// TIA Portal V16 export
// export: Created 2020-03-06T18:52:04.6869857Z, ExportSetting WithDefaults, DisplayName Totally Integrated Automation Portal, DisplayVersion V16, DisplayName TIA Portal Version Control Interface, DisplayVersion V16, DisplayName TIA Portal Openness, DisplayVersion V16, DisplayName TIA Portal Teamcenter Gateway, DisplayVersion V16, DisplayName SINAMICS Startdrive Advanced, DisplayVersion V16 Update 1, DisplayName SINAMICS Startdrive G130, G150, S120, S150, SINAMICS MV, S210, DisplayVersion V16 Update 1, DisplayName SINAMICS Startdrive G110M, G120, G120C, G120D, G120P, DisplayVersion V16 Update 1, DisplayName STEP 7 Professional, DisplayVersion V16, DisplayName STEP 7 Safety, DisplayVersion V16, DisplayName WinCC Professional, DisplayVersion V16
FUNCTION_BLOCK "Median 3RR"   // FB871, LAD
{ S7_Optimized_Access := 'TRUE' }
VERSION : 0.3
// stored: AutoNumber false, IsIECCheckEnabled false, IsRetainMemResEnabled false, MemoryReserve 100, SetENOAutomatically false, UDAEnableTagReadback false
   VAR_INPUT
      V1 { ExternalAccessible := 'False'; ExternalVisible := 'False'; ExternalWritable := 'False'} : Real;   // Value 1 REAL
      V2 { ExternalAccessible := 'False'; ExternalVisible := 'False'; ExternalWritable := 'False'} : Real;   // Value 2 REAL
      V3 { ExternalAccessible := 'False'; ExternalVisible := 'False'; ExternalWritable := 'False'} : Real;   // Value 3 REAL
   END_VAR
   VAR_OUTPUT
      MV { ExternalAccessible := 'False'; ExternalVisible := 'False'; ExternalWritable := 'False'} : Real;   // Middle Value
      DGA { ExternalAccessible := 'False'; ExternalVisible := 'False'; ExternalWritable := 'False'} : Bool;   // Deviation General Alarm
      LGA { ExternalAccessible := 'False'; ExternalVisible := 'False'; ExternalWritable := 'False'} : Bool;   // Limit General Alarm
      Spare { ExternalAccessible := 'False'; ExternalVisible := 'False'; ExternalWritable := 'False'} : Bool;   // Spare
   END_VAR
   VAR
      Config : Struct
         DL : Real;   // Deviation Limit
         GL : Real;   // Global Limit
         GH : Real := 1.0;   // Global Hysteresis
         Limits : Struct
            HH : Real;   // High High
            H : Real;   // High
            L : Real;   // Low
            LL : Real;   // Low Low
         END_STRUCT;
         Hysteresis : Struct
            HH : Real;   // High High
            H : Real;   // High
            L : Real;   // Low
            LL : Real;   // Low Low
         END_STRUCT;
      END_STRUCT;
      Status : Struct
         MV : Real;   // Median Value
         HV : Real;   // Highest Value
         LV : Real;   // Lowest Value
         AV : Real;   // Average Value
         V1D : Real;   // Value 1 Deviation
         V2D : Real;   // Value 2 Deviation
         V3D : Real;   // Value 3 Deviation
         V1MV : Bool;   // Value 1 is the Middle Value
         V2MV : Bool;   // Value 2 is the Middle Value
         V3MV : Bool;   // Value 3 is the Middle Value
      END_STRUCT;
      Alarms : Struct
         VHH : Bool;   // Value High High Alarm
         VH : Bool;   // Value High Alarm
         VL : Bool;   // Value Low Alarm
         VLL : Bool;   // Value Low Low Alarm
         V1OD : Bool;   // Value 1 Over Deviation
         V2OD : Bool;   // Value 2 Over Deviation
         V3OD : Bool;   // Value 3 Over Deviation
      END_STRUCT;
      HHA { ExternalAccessible := 'False'; ExternalVisible := 'False'; ExternalWritable := 'False'} : "HLR";   // High High Alarm
      HA { ExternalAccessible := 'False'; ExternalVisible := 'False'; ExternalWritable := 'False'} : "HLR";   // High Alarm
      LA { ExternalAccessible := 'False'; ExternalVisible := 'False'; ExternalWritable := 'False'} : "LLR";   // Low Alarm
      LLA { ExternalAccessible := 'False'; ExternalVisible := 'False'; ExternalWritable := 'False'} : "LLR";   // Low Low Alarm
      V1DL { ExternalAccessible := 'False'; ExternalVisible := 'False'; ExternalWritable := 'False'} : "HLR";   // Value 1 Deviation Limit
      V2DL { ExternalAccessible := 'False'; ExternalVisible := 'False'; ExternalWritable := 'False'} : "HLR";   // Value 2 Deviation Limit
      V3DL { ExternalAccessible := 'False'; ExternalVisible := 'False'; ExternalWritable := 'False'} : "HLR";   // Value 3 Deviation Limit
   END_VAR
   VAR_TEMP
      ME1 : Real;   // Math Equation 1
      ME2 : Real;   // Math Equation 2
      LDV : Real;   // Lowest Deviation Value
      V1DNA : Real;   // Value 1 Deviation Not Absolute
      V2DNA : Real;   // Value 2 Deviation Not Absolute
      V3DNA : Real;   // Value 3 Deviation Not Absolute
      V1DA : Real;   // Value 1 Deviation Absolute
      V2DA : Real;   // Value 2 Deviation Absolute
      V3DA : Real;   // Value 3 Deviation Absolute
      V1MDA : Real;   // Value 1 Median Deviation Absolute
      V2MDA : Real;   // Value 2 Median Deviation Absolute
      V3MDA : Real;   // Value 3 Median Deviation Absolute
   END_VAR
   VAR_TEMP   // added for the SCL form of the ladder/FBD networks
      _w1 : Bool;
   END_VAR
BEGIN

REGION Network 1: Highest Value
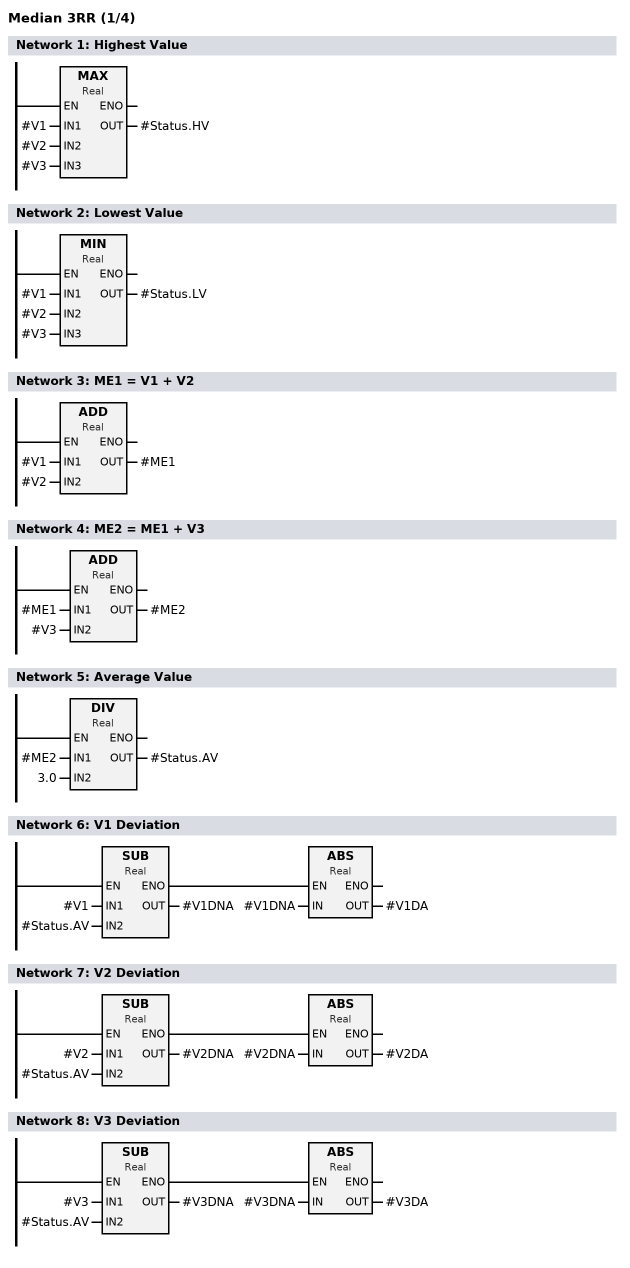
   RUNG wire#powerrail
      { S7_Templates := "[card := 3, value_type := Real]" } MAX(in1 := #V1, in2 := #V2, in3 := #V3, out => #Status.HV)
   END_RUNG
   // the same network as SCL:
   #Status.HV := MAX(IN1 := #V1, IN2 := #V2, IN3 := #V3);
END_REGION

REGION Network 2: Lowest Value
   RUNG wire#powerrail
      { S7_Templates := "[card := 3, value_type := Real]" } MIN(in1 := #V1, in2 := #V2, in3 := #V3, out => #Status.LV)
   END_RUNG
   // the same network as SCL:
   #Status.LV := MIN(IN1 := #V1, IN2 := #V2, IN3 := #V3);
END_REGION

REGION Network 3: ME1 = V1 + V2
   RUNG wire#powerrail
      { S7_Templates := "SrcType := Real"; S7_GenerateENO := "TRUE" } Add(in1 := #V1, in2 := #V2, out => #ME1)
   END_RUNG
   // the same network as SCL:
   #ME1 := #V1 + #V2;
END_REGION

REGION Network 4: ME2 = ME1 + V3
   RUNG wire#powerrail
      { S7_Templates := "SrcType := Real"; S7_GenerateENO := "TRUE" } Add(in1 := #ME1, in2 := #V3, out => #ME2)
   END_RUNG
   // the same network as SCL:
   #ME2 := #ME1 + #V3;
END_REGION

REGION Network 5: Average Value
   RUNG wire#powerrail
      { S7_Templates := "SrcType := Real"; S7_GenerateENO := "TRUE" } Div(in1 := #ME2, in2 := 3.0, out => #Status.AV)
   END_RUNG
   // the same network as SCL:
   #Status.AV := #ME2 / 3.0;
END_REGION

REGION Network 6: V1 Deviation
   RUNG wire#powerrail
      { S7_Templates := "SrcType := Real"; S7_GenerateENO := "TRUE" } Sub(in1 := #V1, in2 := #Status.AV, out => #V1DNA)
      { S7_Templates := "SrcType := Real"; S7_GenerateENO := "TRUE" } Abs(in := #V1DNA, out => #V1DA)
   END_RUNG
   // the same network as SCL:
   // ENO of a box is taken as its EN; it also drops when the box reports an error
   #V1DNA := #V1 - #Status.AV;
   #V1DA := ABS(#V1DNA);
END_REGION

REGION Network 7: V2 Deviation
   RUNG wire#powerrail
      { S7_Templates := "SrcType := Real"; S7_GenerateENO := "TRUE" } Sub(in1 := #V2, in2 := #Status.AV, out => #V2DNA)
      { S7_Templates := "SrcType := Real"; S7_GenerateENO := "TRUE" } Abs(in := #V2DNA, out => #V2DA)
   END_RUNG
   // the same network as SCL:
   // ENO of a box is taken as its EN; it also drops when the box reports an error
   #V2DNA := #V2 - #Status.AV;
   #V2DA := ABS(#V2DNA);
END_REGION

REGION Network 8: V3 Deviation
   RUNG wire#powerrail
      { S7_Templates := "SrcType := Real"; S7_GenerateENO := "TRUE" } Sub(in1 := #V3, in2 := #Status.AV, out => #V3DNA)
      { S7_Templates := "SrcType := Real"; S7_GenerateENO := "TRUE" } Abs(in := #V3DNA, out => #V3DA)
   END_RUNG
   // the same network as SCL:
   // ENO of a box is taken as its EN; it also drops when the box reports an error
   #V3DNA := #V3 - #Status.AV;
   #V3DA := ABS(#V3DNA);
END_REGION

REGION Network 9
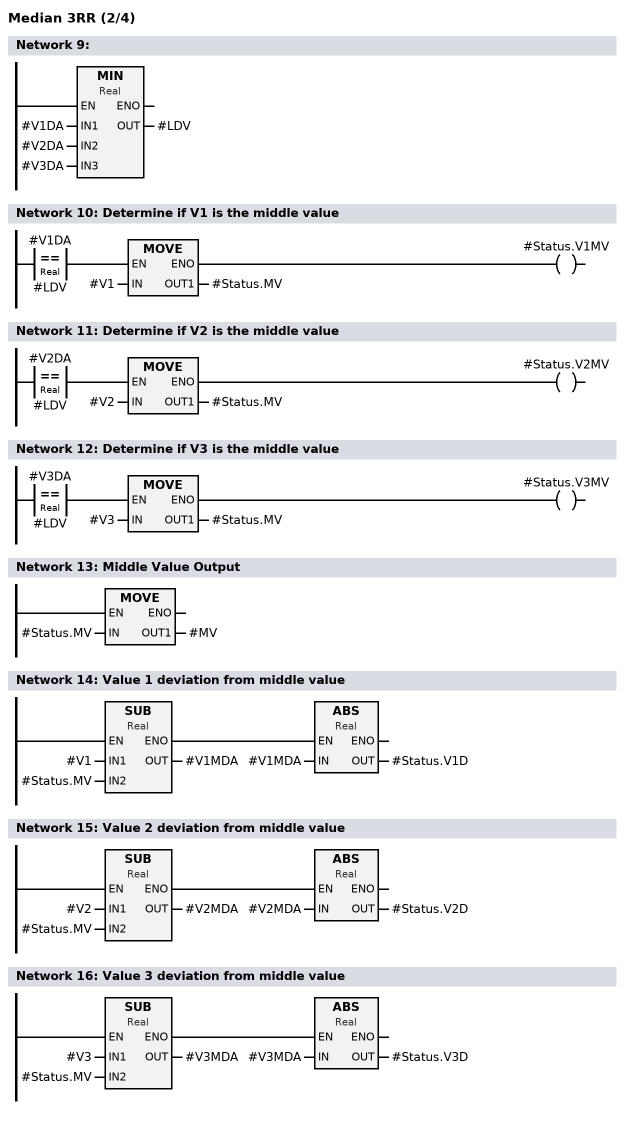
   RUNG wire#powerrail
      { S7_Templates := "[card := 3, value_type := Real]" } MIN(in1 := #V1DA, in2 := #V2DA, in3 := #V3DA, out => #LDV)
   END_RUNG
   // the same network as SCL:
   #LDV := MIN(IN1 := #V1DA, IN2 := #V2DA, IN3 := #V3DA);
END_REGION

REGION Network 10: Determine if V1 is the middle value
   RUNG wire#powerrail
      { S7_Templates := "SrcType := Real" } EQ_Contact(in1 := #V1DA, in2 := #LDV)
      { S7_GenerateENO := "TRUE" } Move(in := #V1, out1 => #Status.MV)
      Coil( #Status.V1MV )
   END_RUNG
   // the same network as SCL:
   // ENO of a box is taken as its EN; it also drops when the box reports an error
   #_w1 := #V1DA = #LDV;
   IF #_w1 THEN #Status.MV := #V1; END_IF;
   #Status.V1MV := #_w1;
END_REGION

REGION Network 11: Determine if V2 is the middle value
   RUNG wire#powerrail
      { S7_Templates := "SrcType := Real" } EQ_Contact(in1 := #V2DA, in2 := #LDV)
      { S7_GenerateENO := "TRUE" } Move(in := #V2, out1 => #Status.MV)
      Coil( #Status.V2MV )
   END_RUNG
   // the same network as SCL:
   // ENO of a box is taken as its EN; it also drops when the box reports an error
   #_w1 := #V2DA = #LDV;
   IF #_w1 THEN #Status.MV := #V2; END_IF;
   #Status.V2MV := #_w1;
END_REGION

REGION Network 12: Determine if V3 is the middle value
   RUNG wire#powerrail
      { S7_Templates := "SrcType := Real" } EQ_Contact(in1 := #V3DA, in2 := #LDV)
      { S7_GenerateENO := "TRUE" } Move(in := #V3, out1 => #Status.MV)
      Coil( #Status.V3MV )
   END_RUNG
   // the same network as SCL:
   // ENO of a box is taken as its EN; it also drops when the box reports an error
   #_w1 := #V3DA = #LDV;
   IF #_w1 THEN #Status.MV := #V3; END_IF;
   #Status.V3MV := #_w1;
END_REGION

REGION Network 13: Middle Value Output
   RUNG wire#powerrail
      { S7_GenerateENO := "TRUE" } Move(in := #Status.MV, out1 => #MV)
   END_RUNG
   // the same network as SCL:
   #MV := #Status.MV;
END_REGION

REGION Network 14: Value 1 deviation from middle value
   RUNG wire#powerrail
      { S7_Templates := "SrcType := Real"; S7_GenerateENO := "TRUE" } Sub(in1 := #V1, in2 := #Status.MV, out => #V1MDA)
      { S7_Templates := "SrcType := Real"; S7_GenerateENO := "TRUE" } Abs(in := #V1MDA, out => #Status.V1D)
   END_RUNG
   // the same network as SCL:
   // ENO of a box is taken as its EN; it also drops when the box reports an error
   #V1MDA := #V1 - #Status.MV;
   #Status.V1D := ABS(#V1MDA);
END_REGION

REGION Network 15: Value 2 deviation from middle value
   RUNG wire#powerrail
      { S7_Templates := "SrcType := Real"; S7_GenerateENO := "TRUE" } Sub(in1 := #V2, in2 := #Status.MV, out => #V2MDA)
      { S7_Templates := "SrcType := Real"; S7_GenerateENO := "TRUE" } Abs(in := #V2MDA, out => #Status.V2D)
   END_RUNG
   // the same network as SCL:
   // ENO of a box is taken as its EN; it also drops when the box reports an error
   #V2MDA := #V2 - #Status.MV;
   #Status.V2D := ABS(#V2MDA);
END_REGION

REGION Network 16: Value 3 deviation from middle value
   RUNG wire#powerrail
      { S7_Templates := "SrcType := Real"; S7_GenerateENO := "TRUE" } Sub(in1 := #V3, in2 := #Status.MV, out => #V3MDA)
      { S7_Templates := "SrcType := Real"; S7_GenerateENO := "TRUE" } Abs(in := #V3MDA, out => #Status.V3D)
   END_RUNG
   // the same network as SCL:
   // ENO of a box is taken as its EN; it also drops when the box reports an error
   #V3MDA := #V3 - #Status.MV;
   #Status.V3D := ABS(#V3MDA);
END_REGION

REGION Network 17: Use Global Limit Value if GL is > 0
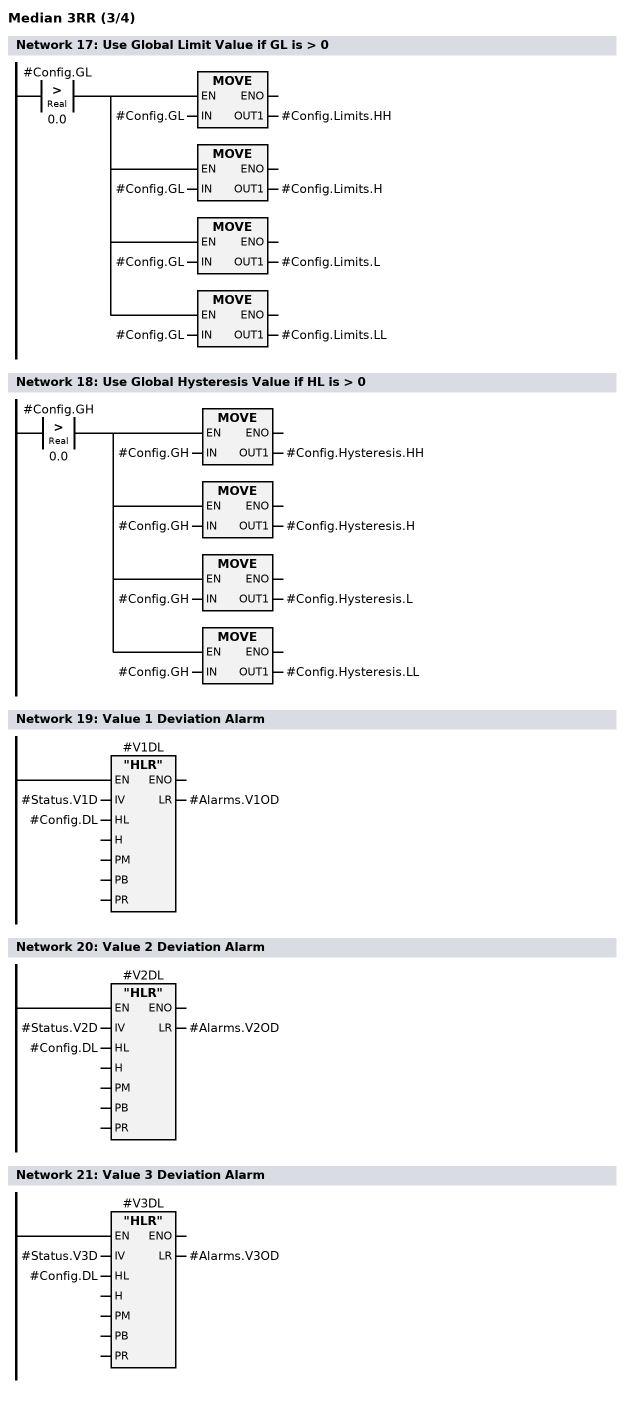
   RUNG wire#powerrail
      { S7_Templates := "SrcType := Real" } GT_Contact(in1 := #Config.GL, in2 := 0.0)
      wire#w1
      { S7_GenerateENO := "TRUE" } Move(in := #Config.GL, out1 => #Config.Limits.HH)
   END_RUNG
   RUNG wire#w1
      { S7_GenerateENO := "TRUE" } Move(in := #Config.GL, out1 => #Config.Limits.H)
   END_RUNG
   RUNG wire#w1
      { S7_GenerateENO := "TRUE" } Move(in := #Config.GL, out1 => #Config.Limits.L)
   END_RUNG
   RUNG wire#w1
      { S7_GenerateENO := "TRUE" } Move(in := #Config.GL, out1 => #Config.Limits.LL)
   END_RUNG
   // the same network as SCL:
   IF #Config.GL > 0.0 THEN
       #Config.Limits.HH := #Config.GL;
       #Config.Limits.H := #Config.GL;
       #Config.Limits.L := #Config.GL;
       #Config.Limits.LL := #Config.GL;
   END_IF;
END_REGION

REGION Network 18: Use Global Hysteresis Value if HL is > 0
   RUNG wire#powerrail
      { S7_Templates := "SrcType := Real" } GT_Contact(in1 := #Config.GH, in2 := 0.0)
      wire#w1
      { S7_GenerateENO := "TRUE" } Move(in := #Config.GH, out1 => #Config.Hysteresis.HH)
   END_RUNG
   RUNG wire#w1
      { S7_GenerateENO := "TRUE" } Move(in := #Config.GH, out1 => #Config.Hysteresis.H)
   END_RUNG
   RUNG wire#w1
      { S7_GenerateENO := "TRUE" } Move(in := #Config.GH, out1 => #Config.Hysteresis.L)
   END_RUNG
   RUNG wire#w1
      { S7_GenerateENO := "TRUE" } Move(in := #Config.GH, out1 => #Config.Hysteresis.LL)
   END_RUNG
   // the same network as SCL:
   IF #Config.GH > 0.0 THEN
       #Config.Hysteresis.HH := #Config.GH;
       #Config.Hysteresis.H := #Config.GH;
       #Config.Hysteresis.L := #Config.GH;
       #Config.Hysteresis.LL := #Config.GH;
   END_IF;
END_REGION

REGION Network 19: Value 1 Deviation Alarm
   RUNG wire#powerrail
      #V1DL(IV := #Status.V1D, HL := #Config.DL, H :=, PM :=, PB :=, PR :=, LR => #Alarms.V1OD)
   END_RUNG
   // the same network as SCL:
   #V1DL(IV := #Status.V1D, HL := #Config.DL, LR => #Alarms.V1OD);   // "HLR"
END_REGION

REGION Network 20: Value 2 Deviation Alarm
   RUNG wire#powerrail
      #V2DL(IV := #Status.V2D, HL := #Config.DL, H :=, PM :=, PB :=, PR :=, LR => #Alarms.V2OD)
   END_RUNG
   // the same network as SCL:
   #V2DL(IV := #Status.V2D, HL := #Config.DL, LR => #Alarms.V2OD);   // "HLR"
END_REGION

REGION Network 21: Value 3 Deviation Alarm
   RUNG wire#powerrail
      #V3DL(IV := #Status.V3D, HL := #Config.DL, H :=, PM :=, PB :=, PR :=, LR => #Alarms.V3OD)
   END_RUNG
   // the same network as SCL:
   #V3DL(IV := #Status.V3D, HL := #Config.DL, LR => #Alarms.V3OD);   // "HLR"
END_REGION

REGION Network 22: Deviation General Alarm
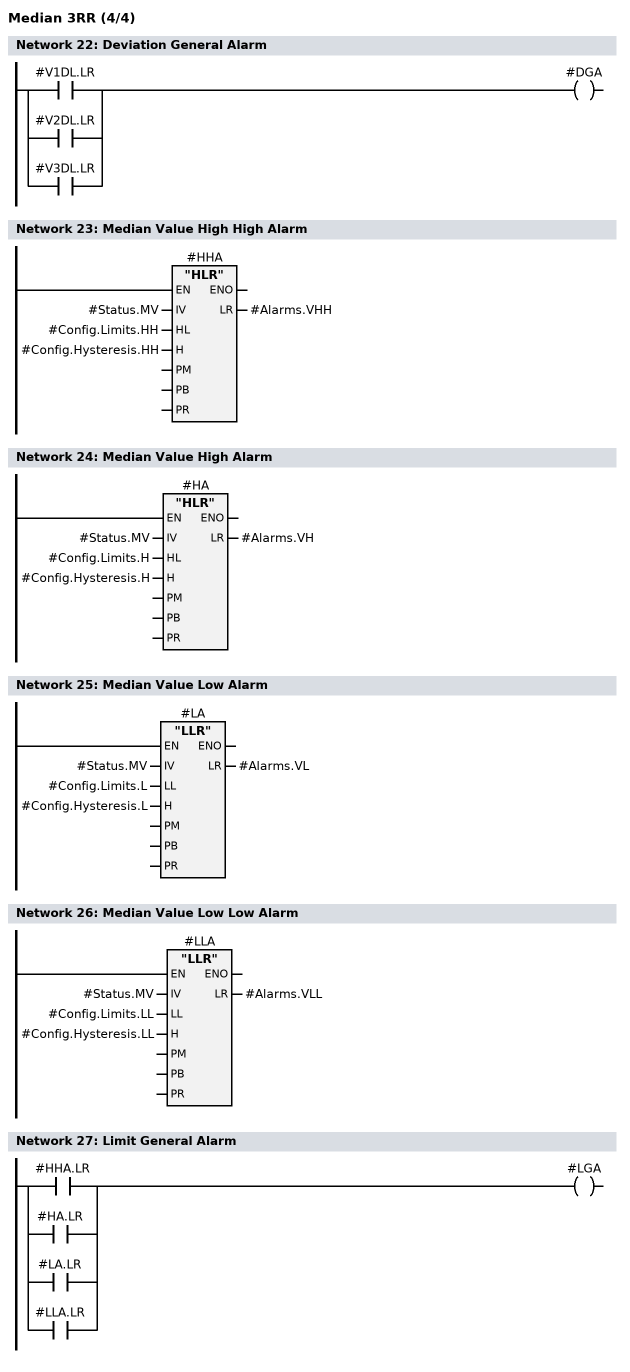
   RUNG wire#powerrail
      Contact( #V1DL.LR )
      wire#w1
      Coil( #DGA )
   END_RUNG
   RUNG wire#powerrail
      Contact( #V2DL.LR )
   END_RUNG wire#w1
   RUNG wire#powerrail
      Contact( #V3DL.LR )
   END_RUNG wire#w1
   // the same network as SCL:
   #DGA := #V1DL.LR OR #V2DL.LR OR #V3DL.LR;
END_REGION

REGION Network 23: Median Value High High Alarm
   RUNG wire#powerrail
      #HHA(IV := #Status.MV, HL := #Config.Limits.HH, H := #Config.Hysteresis.HH, PM :=, PB :=, PR :=, LR => #Alarms.VHH)
   END_RUNG
   // the same network as SCL:
   #HHA(IV := #Status.MV, HL := #Config.Limits.HH, H := #Config.Hysteresis.HH, LR => #Alarms.VHH);   // "HLR"
END_REGION

REGION Network 24: Median Value High Alarm
   RUNG wire#powerrail
      #HA(IV := #Status.MV, HL := #Config.Limits.H, H := #Config.Hysteresis.H, PM :=, PB :=, PR :=, LR => #Alarms.VH)
   END_RUNG
   // the same network as SCL:
   #HA(IV := #Status.MV, HL := #Config.Limits.H, H := #Config.Hysteresis.H, LR => #Alarms.VH);   // "HLR"
END_REGION

REGION Network 25: Median Value Low Alarm
   RUNG wire#powerrail
      #LA(IV := #Status.MV, LL := #Config.Limits.L, H := #Config.Hysteresis.L, PM :=, PB :=, PR :=, LR => #Alarms.VL)
   END_RUNG
   // the same network as SCL:
   #LA(IV := #Status.MV, LL := #Config.Limits.L, H := #Config.Hysteresis.L, LR => #Alarms.VL);   // "LLR"
END_REGION

REGION Network 26: Median Value Low Low Alarm
   RUNG wire#powerrail
      #LLA(IV := #Status.MV, LL := #Config.Limits.LL, H := #Config.Hysteresis.LL, PM :=, PB :=, PR :=, LR => #Alarms.VLL)
   END_RUNG
   // the same network as SCL:
   #LLA(IV := #Status.MV, LL := #Config.Limits.LL, H := #Config.Hysteresis.LL, LR => #Alarms.VLL);   // "LLR"
END_REGION

REGION Network 27: Limit General Alarm
   RUNG wire#powerrail
      Contact( #HHA.LR )
      wire#w1
      Coil( #LGA )
   END_RUNG
   RUNG wire#powerrail
      Contact( #HA.LR )
   END_RUNG wire#w1
   RUNG wire#powerrail
      Contact( #LA.LR )
   END_RUNG wire#w1
   RUNG wire#powerrail
      Contact( #LLA.LR )
   END_RUNG wire#w1
   // the same network as SCL:
   #LGA := #HHA.LR OR #HA.LR OR #LA.LR OR #LLA.LR;
END_REGION
END_FUNCTION_BLOCK
